FUNCTION_BLOCK PicknPlace (* Basic Function Block Type *)
  (* Standard: 61499-2 *)
  (* Version 0.0, 2015-03-26, 4DIAC-IDE, 4DIAC-Consortium *)
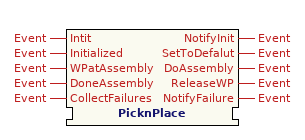
  EVENT_INPUT
    Intit;
    Initialized;
    WPatAssembly;
    DoneAssembly;
    CollectFailures;
  END_EVENT
  EVENT_OUTPUT
    NotifyInit;
    SetToDefalut; (* Initialization Confirm *)
    DoAssembly;
    ReleaseWP;
    NotifyFailure;
  END_EVENT
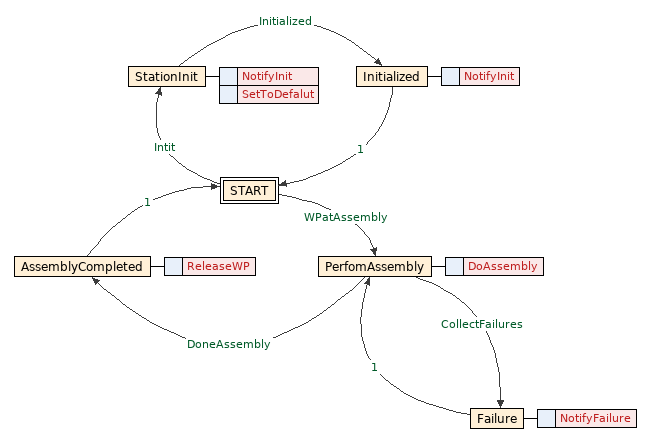
  EC_STATES
    START; (* Initial State *)
    StationInit : -> NotifyInit, -> SetToDefalut;
    PerfomAssembly : -> DoAssembly;
    AssemblyCompleted : -> ReleaseWP;
    Failure : -> NotifyFailure;
    Initialized : -> NotifyInit;
  END_STATES
  EC_TRANSITIONS
    START TO StationInit := Intit;
    PerfomAssembly TO AssemblyCompleted := DoneAssembly;
    START TO PerfomAssembly := WPatAssembly;
    AssemblyCompleted TO START := 1;
    Failure TO PerfomAssembly := 1;
    PerfomAssembly TO Failure := CollectFailures;
    Initialized TO START := 1;
    StationInit TO Initialized := Initialized;
  END_TRANSITIONS
  ALGORITHM INIT IN ST: (* Initialization algorithm *)

  END_ALGORITHM
  ALGORITHM REQ IN ST: (* Normally executed algorithm *)

  END_ALGORITHM
END_FUNCTION_BLOCK
